// Mitsubishi GX Works2 project: De05   PLC: FX2N/FX2NC

PROGRAM MAIN
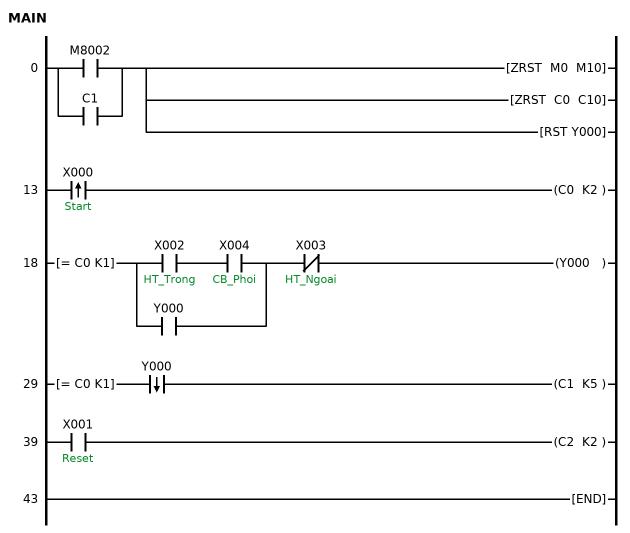
0     LD      M8002
      OR      C1
      ZRST    M0 M10
      ZRST    C0 C10
      RST     Y000
13    LDP     X000  ; Start
      OUT     C0 K2
18    LD=     C0 K1
      LD      X002  ; HT_Trong
      AND     X004  ; CB_Phoi
      OR      Y000
      ANB
      ANI     X003  ; HT_Ngoai
      OUT     Y000
29    LD=     C0 K1
      ANDF    Y000
      OUT     C1 K5
39    LD      X001  ; Reset
      OUT     C2 K2
43    END
END_PROGRAM
